VISUALIZATION VISU_State_gray_yellow  // 12x17
VAR_IN_OUT
	state : BOOL;
END_VAR
    Ellipse (0,5 10x10), colour toggle: state
END_VISUALIZATION

(* stored: Version 1.1.0.1, ProductVersion 3.1.4018.5
   Visu VISU_State_gray_yellow: Id {8f104871-8951-4a59-b5f4-b924179547e9} *)
